{attribute 'qualified_only'}
VAR_GLOBAL
    fbArbiter: FB_Arbiter;
    fbFastFaultOutput1: FB_HardwareFFOutput;
    fbFastFaultOutput2: FB_HardwareFFOutput;

// MPS fault reset, add temporarily to use FB_MPA
     xFastFaultReset :   BOOL;
END_VAR

(* stored: Version 1.1.0.1, ProductVersion 3.1.4022.18
   GVL PMPS: Id {7ed09a37-cf90-49ac-9e4a-5fe59e47274f} *)
